(* Logix 5000 project; controller Google vendor 1 type 14 code 151 rev 31.11; software revision 31.00; part 4 of 5 *)
(* tags used below, declared in another part *)
   Infeed_Active : BOOL;
   L1_Clear_Out : BOOL;
   L1_Empty_Delay : TIMER;
   L1_Full_Delay : TIMER;
   L1_Zone1 : Zone_Data;
   L1_Zone1_2_ProdCode : DINT;
   L1_Zone1_2_ProdName : STRING;
   L1_Zone1_FWD : BOOL;
   L1_Zone1_PE : BOOL;
   L1_Zone1_ProdCode : DINT;
   L1_Zone1_ProdName : STRING;
   L1_Zone1_REV : BOOL;
   L1_Zone2 : Zone_Data;
   L1_Zone2_3_ProdCode : DINT;
   L1_Zone2_3_ProdName : STRING;
   L1_Zone2_FWD : BOOL;
   L1_Zone2_PE : BOOL;
   L1_Zone2_ProdCode : DINT;
   L1_Zone2_ProdName : STRING;
   L1_Zone2_REV : BOOL;
   L1_Zone3 : Zone_Data;
   L1_Zone3_4_ProdCode : DINT;
   L1_Zone3_4_ProdName : STRING;
   L1_Zone3_FWD : BOOL;
   L1_Zone3_PE : BOOL;
   L1_Zone3_ProdCode : DINT;
   L1_Zone3_ProdName : STRING;
   L1_Zone3_REV : BOOL;
   L1_Zone4 : End_Zone_Data;
   L1_Zone4_FWD : BOOL;
   L1_Zone4_PE : BOOL;
   L1_Zone4_ProdCode : DINT;
   L1_Zone4_ProdName : STRING;
   L1_Zone4_REV : BOOL;
   L1_Zone_Timeout : TIMER[8];
   L2_Empty_Delay : TIMER;
   L2_Full_Delay : TIMER;
   L2_Z1_Outfeed : BOOL;
   L2_Z2_Outfeed : BOOL;
   L2_Z3_Outfeed : BOOL;
   L2_Z4_Outfeed : BOOL;
   L2_Zone1 : Zone_Data;
   L2_Zone1_2_ProdCode : DINT;
   L2_Zone1_2_ProdName : STRING;
   L2_Zone1_FWD : BOOL;
   L2_Zone1_PE : BOOL;
   L2_Zone1_ProdCode : DINT;
   L2_Zone1_ProdName : STRING;
   L2_Zone1_REV : BOOL;
   L2_Zone2 : Zone_Data;
   L2_Zone2_3_ProdCode : DINT;
   L2_Zone2_3_ProdName : STRING;
   L2_Zone2_FWD : BOOL;
   L2_Zone2_PE : BOOL;
   L2_Zone2_ProdCode : DINT;
   L2_Zone2_ProdName : STRING;
   L2_Zone2_REV : BOOL;
   L2_Zone3 : Zone_Data;
   L2_Zone3_4_ProdCode : DINT;
   L2_Zone3_4_ProdName : STRING;
   L2_Zone3_FWD : BOOL;
   L2_Zone3_PE : BOOL;
   L2_Zone3_ProdCode : DINT;
   L2_Zone3_ProdName : STRING;
   L2_Zone3_REV : BOOL;
   L2_Zone4 : End_Zone_Data;
   L2_Zone4_FWD : BOOL;
   L2_Zone4_PE : BOOL;
   L2_Zone4_ProdCode : DINT;
   L2_Zone4_ProdName : STRING;
   L2_Zone4_REV : BOOL;
   L2_Zone_Timeout : TIMER[8];
   L3_Empty_Delay : TIMER;
   L3_Full_Delay : TIMER;
   L3_Z1_Outfeed : BOOL;
   L3_Z2_Outfeed : BOOL;
   L3_Z3_Outfeed : BOOL;
   L3_Z4_Outfeed : BOOL;
   L3_Zone1 : Zone_Data;
   L3_Zone1_2_ProdCode : DINT;
   L3_Zone1_2_ProdName : STRING;
   L3_Zone1_FWD : BOOL;
   L3_Zone1_PE : BOOL;
   L3_Zone1_ProdCode : DINT;
   L3_Zone1_ProdName : STRING;
   L3_Zone1_REV : BOOL;
   L3_Zone2 : Zone_Data;
   L3_Zone2_3_ProdCode : DINT;
   L3_Zone2_3_ProdName : STRING;
   L3_Zone2_FWD : BOOL;
   L3_Zone2_PE : BOOL;
   L3_Zone2_ProdCode : DINT;
   L3_Zone2_ProdName : STRING;
   L3_Zone2_REV : BOOL;
   L3_Zone3 : Zone_Data;
   L3_Zone3_4_ProdCode : DINT;
   L3_Zone3_4_ProdName : STRING;
   L3_Zone3_FWD : BOOL;
   L3_Zone3_PE : BOOL;
   L3_Zone3_ProdCode : DINT;
   L3_Zone3_ProdName : STRING;
   L3_Zone3_REV : BOOL;
   L3_Zone4 : End_Zone_Data;
   L3_Zone4_FWD : BOOL;
   L3_Zone4_PE : BOOL;
   L3_Zone4_ProdCode : DINT;
   L3_Zone4_ProdName : STRING;
   L3_Zone4_REV : BOOL;
   L3_Zone_Timeout : TIMER[8];
   L4_Empty_Delay : TIMER;
   L4_Full_Delay : TIMER;
   L4_Z1_Outfeed : BOOL;
   L4_Z2_Outfeed : BOOL;
   L4_Z3_Outfeed : BOOL;
   L4_Z4_Outfeed : BOOL;
   L4_Zone1 : Zone_Data;
   L4_Zone1_2_ProdCode : DINT;
   L4_Zone1_2_ProdName : STRING;
   L4_Zone1_FWD : BOOL;
   L4_Zone1_PE : BOOL;
   L4_Zone1_ProdCode : DINT;
   L4_Zone1_ProdName : STRING;
   L4_Zone1_REV : BOOL;
   L4_Zone2 : Zone_Data;
   L4_Zone2_3_ProdCode : DINT;
   L4_Zone2_3_ProdName : STRING;
   L4_Zone2_FWD : BOOL;
   L4_Zone2_PE : BOOL;
   L4_Zone2_ProdCode : DINT;
   L4_Zone2_ProdName : STRING;
   L4_Zone2_REV : BOOL;
   L4_Zone3 : Zone_Data;
   L4_Zone3_4_ProdCode : DINT;
   L4_Zone3_4_ProdName : STRING;
   L4_Zone3_FWD : BOOL;
   L4_Zone3_PE : BOOL;
   L4_Zone3_ProdCode : DINT;
   L4_Zone3_ProdName : STRING;
   L4_Zone3_REV : BOOL;
   L4_Zone4 : End_Zone_Data;
   L4_Zone4_FWD : BOOL;
   L4_Zone4_PE : BOOL;
   L4_Zone4_ProdCode : DINT;
   L4_Zone4_ProdName : STRING;
   L4_Zone4_REV : BOOL;
   L4_Zone_Timeout : TIMER[8];
   Level_1_Empty : BOOL;
   Level_1_Full : BOOL;
   Level_2_Empty : BOOL;
   Level_2_Full : BOOL;
   Level_3_Empty : BOOL;
   Level_3_Full : BOOL;
   Level_4_Empty : BOOL;
   Level_4_Full : BOOL;
   Lift_Current_Level : DINT;
   Lift_Required_Level : DINT;
   Lift_Zone : Lift_Zone_Data;
   LiftZone_FWD : BOOL;
   LiftZoneDownstream_ProdCode : DINT;
   LiftZoneDownstream_ProdName : STRING;
   Outfeed_Active : BOOL;
   Sort_Number : DINT;
(* MainProgram, continued *)

ROUTINE R09_L1_Conveyor   (* ladder *)
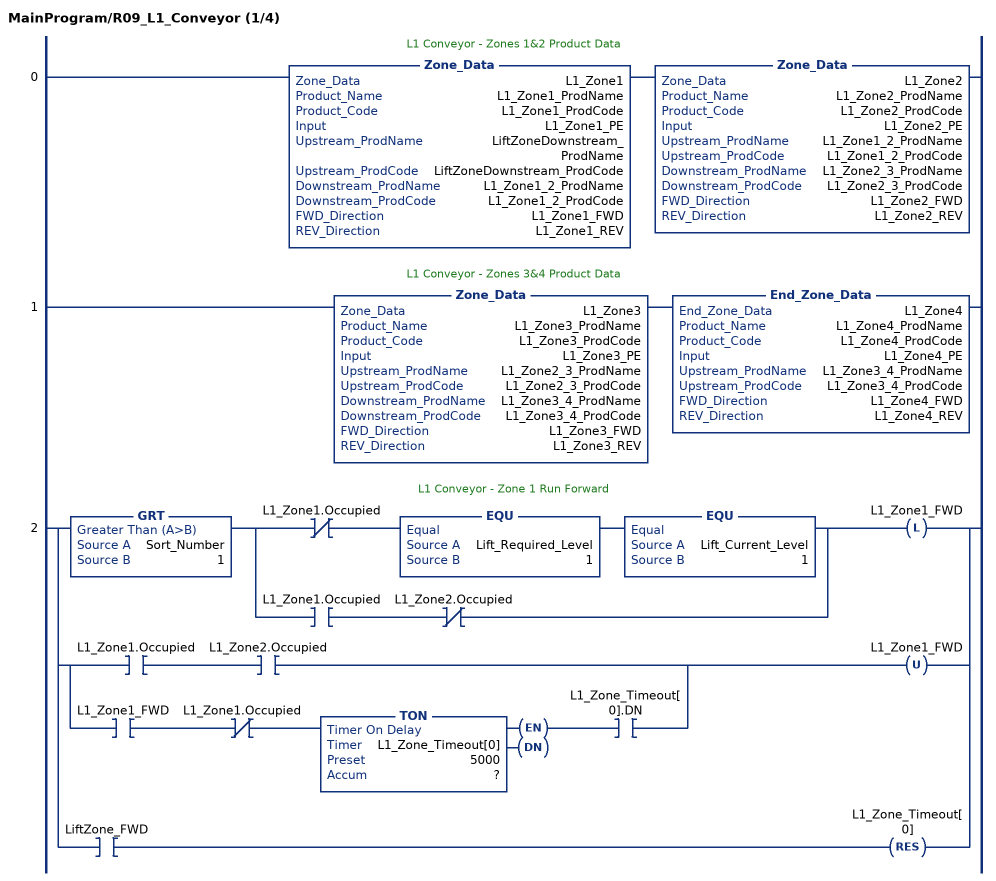
   // L1 Conveyor - Zones 1&2 Product Data
   0: Zone_Data(L1_Zone1,L1_Zone1_ProdName,L1_Zone1_ProdCode,L1_Zone1_PE,LiftZoneDownstream_ProdName,LiftZoneDownstream_ProdCode,L1_Zone1_2_ProdName,L1_Zone1_2_ProdCode,L1_Zone1_FWD,L1_Zone1_REV)Zone_Data(L1_Zone2,L1_Zone2_ProdName,L1_Zone2_ProdCode,L1_Zone2_PE,L1_Zone1_2_ProdName,L1_Zone1_2_ProdCode,L1_Zone2_3_ProdName,L1_Zone2_3_ProdCode,L1_Zone2_FWD,L1_Zone2_REV);
   // L1 Conveyor - Zones 3&4 Product Data
   1: Zone_Data(L1_Zone3,L1_Zone3_ProdName,L1_Zone3_ProdCode,L1_Zone3_PE,L1_Zone2_3_ProdName,L1_Zone2_3_ProdCode,L1_Zone3_4_ProdName,L1_Zone3_4_ProdCode,L1_Zone3_FWD,L1_Zone3_REV)End_Zone_Data(L1_Zone4,L1_Zone4_ProdName,L1_Zone4_ProdCode,L1_Zone4_PE,L1_Zone3_4_ProdName,L1_Zone3_4_ProdCode,L1_Zone4_FWD,L1_Zone4_REV);
   // L1 Conveyor - Zone 1 Run Forward
   2: [GRT(Sort_Number,1) [XIO(L1_Zone1.Occupied) EQU(Lift_Required_Level,1) EQU(Lift_Current_Level,1) ,XIC(L1_Zone1.Occupied) XIO(L1_Zone2.Occupied) ] OTL(L1_Zone1_FWD) ,[XIC(L1_Zone1.Occupied) XIC(L1_Zone2.Occupied) ,XIC(L1_Zone1_FWD) XIO(L1_Zone1.Occupied) TON(L1_Zone_Timeout[0],?,?) XIC(L1_Zone_Timeout[0].DN) ] OTU(L1_Zone1_FWD) ,XIC(LiftZone_FWD) RES(L1_Zone_Timeout[0]) ];
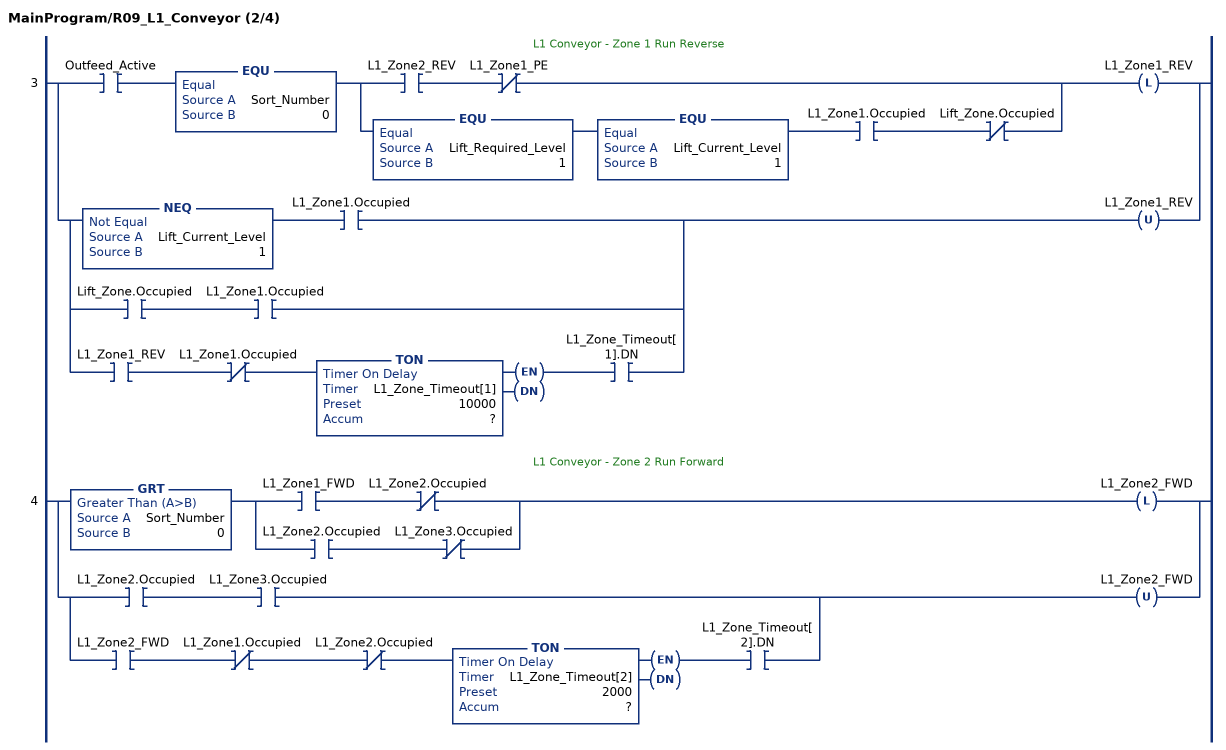
   // L1 Conveyor - Zone 1 Run Reverse
   3: [XIC(Outfeed_Active) EQU(Sort_Number,0) [XIC(L1_Zone2_REV) XIO(L1_Zone1_PE) ,EQU(Lift_Required_Level,1) EQU(Lift_Current_Level,1) XIC(L1_Zone1.Occupied) XIO(Lift_Zone.Occupied) ] OTL(L1_Zone1_REV) ,[NEQ(Lift_Current_Level,1) XIC(L1_Zone1.Occupied) ,XIC(Lift_Zone.Occupied) XIC(L1_Zone1.Occupied) ,XIC(L1_Zone1_REV) XIO(L1_Zone1.Occupied) TON(L1_Zone_Timeout[1],?,?) XIC(L1_Zone_Timeout[1].DN) ] OTU(L1_Zone1_REV) ];
   // L1 Conveyor - Zone 2 Run Forward
   4: [GRT(Sort_Number,0) [XIC(L1_Zone1_FWD) XIO(L1_Zone2.Occupied) ,XIC(L1_Zone2.Occupied) XIO(L1_Zone3.Occupied) ] OTL(L1_Zone2_FWD) ,[XIC(L1_Zone2.Occupied) XIC(L1_Zone3.Occupied) ,XIC(L1_Zone2_FWD) XIO(L1_Zone1.Occupied) XIO(L1_Zone2.Occupied) TON(L1_Zone_Timeout[2],?,?) XIC(L1_Zone_Timeout[2].DN) ] OTU(L1_Zone2_FWD) ];
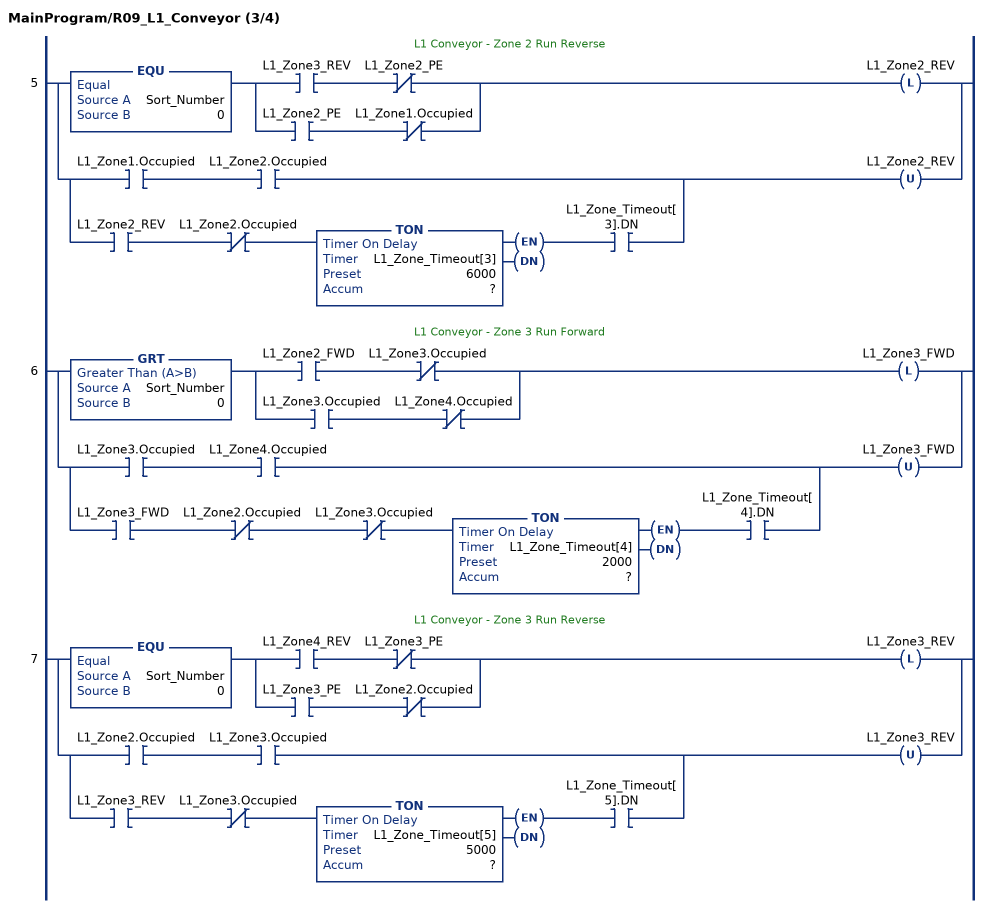
   // L1 Conveyor - Zone 2 Run Reverse
   5: [EQU(Sort_Number,0) [XIC(L1_Zone3_REV) XIO(L1_Zone2_PE) ,XIC(L1_Zone2_PE) XIO(L1_Zone1.Occupied) ] OTL(L1_Zone2_REV) ,[XIC(L1_Zone1.Occupied) XIC(L1_Zone2.Occupied) ,XIC(L1_Zone2_REV) XIO(L1_Zone2.Occupied) TON(L1_Zone_Timeout[3],?,?) XIC(L1_Zone_Timeout[3].DN) ] OTU(L1_Zone2_REV) ];
   // L1 Conveyor - Zone 3 Run Forward
   6: [GRT(Sort_Number,0) [XIC(L1_Zone2_FWD) XIO(L1_Zone3.Occupied) ,XIC(L1_Zone3.Occupied) XIO(L1_Zone4.Occupied) ] OTL(L1_Zone3_FWD) ,[XIC(L1_Zone3.Occupied) XIC(L1_Zone4.Occupied) ,XIC(L1_Zone3_FWD) XIO(L1_Zone2.Occupied) XIO(L1_Zone3.Occupied) TON(L1_Zone_Timeout[4],?,?) XIC(L1_Zone_Timeout[4].DN) ] OTU(L1_Zone3_FWD) ];
   // L1 Conveyor - Zone 3 Run Reverse
   7: [EQU(Sort_Number,0) [XIC(L1_Zone4_REV) XIO(L1_Zone3_PE) ,XIC(L1_Zone3_PE) XIO(L1_Zone2.Occupied) ] OTL(L1_Zone3_REV) ,[XIC(L1_Zone2.Occupied) XIC(L1_Zone3.Occupied) ,XIC(L1_Zone3_REV) XIO(L1_Zone3.Occupied) TON(L1_Zone_Timeout[5],?,?) XIC(L1_Zone_Timeout[5].DN) ] OTU(L1_Zone3_REV) ];
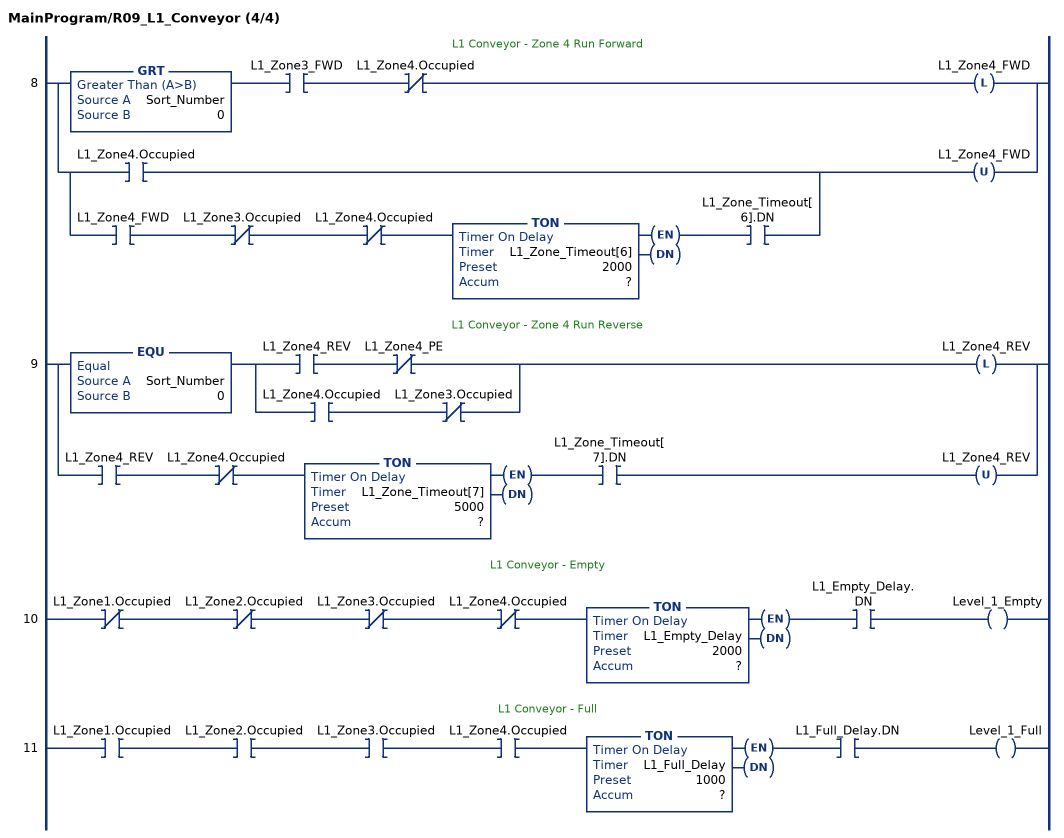
   // L1 Conveyor - Zone 4 Run Forward
   8: [GRT(Sort_Number,0) XIC(L1_Zone3_FWD) XIO(L1_Zone4.Occupied) OTL(L1_Zone4_FWD) ,[XIC(L1_Zone4.Occupied) ,XIC(L1_Zone4_FWD) XIO(L1_Zone3.Occupied) XIO(L1_Zone4.Occupied) TON(L1_Zone_Timeout[6],?,?) XIC(L1_Zone_Timeout[6].DN) ] OTU(L1_Zone4_FWD) ];
   // L1 Conveyor - Zone 4 Run Reverse
   9: [EQU(Sort_Number,0) [XIC(L1_Zone4_REV) XIO(L1_Zone4_PE) ,XIC(L1_Zone4.Occupied) XIO(L1_Zone3.Occupied) ] OTL(L1_Zone4_REV) ,XIC(L1_Zone4_REV) XIO(L1_Zone4.Occupied) TON(L1_Zone_Timeout[7],?,?) XIC(L1_Zone_Timeout[7].DN) OTU(L1_Zone4_REV) ];
   // L1 Conveyor - Empty
   10: XIO(L1_Zone1.Occupied)XIO(L1_Zone2.Occupied)XIO(L1_Zone3.Occupied)XIO(L1_Zone4.Occupied)TON(L1_Empty_Delay,?,?)XIC(L1_Empty_Delay.DN)OTE(Level_1_Empty);
   // L1 Conveyor - Full
   11: XIC(L1_Zone1.Occupied)XIC(L1_Zone2.Occupied)XIC(L1_Zone3.Occupied)XIC(L1_Zone4.Occupied)TON(L1_Full_Delay,?,?)XIC(L1_Full_Delay.DN)OTE(Level_1_Full);
END_ROUTINE

ROUTINE R10_L2_Conveyor   (* ladder *)
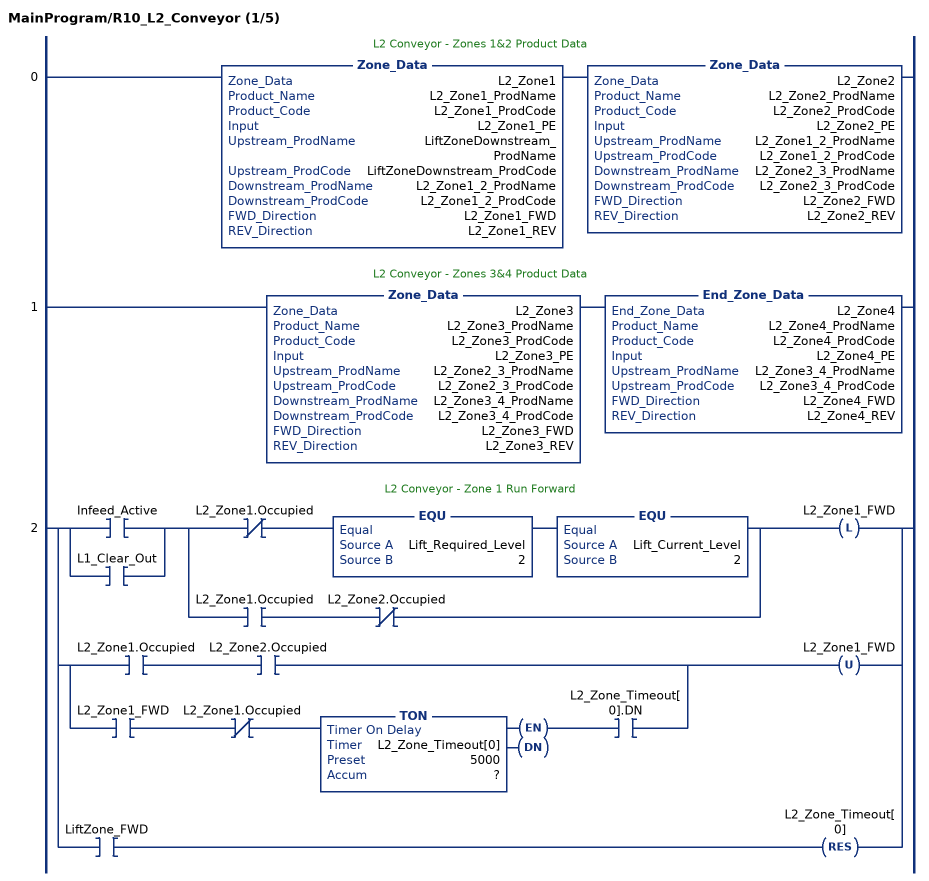
   // L2 Conveyor - Zones 1&2 Product Data
   0: Zone_Data(L2_Zone1,L2_Zone1_ProdName,L2_Zone1_ProdCode,L2_Zone1_PE,LiftZoneDownstream_ProdName,LiftZoneDownstream_ProdCode,L2_Zone1_2_ProdName,L2_Zone1_2_ProdCode,L2_Zone1_FWD,L2_Zone1_REV)Zone_Data(L2_Zone2,L2_Zone2_ProdName,L2_Zone2_ProdCode,L2_Zone2_PE,L2_Zone1_2_ProdName,L2_Zone1_2_ProdCode,L2_Zone2_3_ProdName,L2_Zone2_3_ProdCode,L2_Zone2_FWD,L2_Zone2_REV);
   // L2 Conveyor - Zones 3&4 Product Data
   1: Zone_Data(L2_Zone3,L2_Zone3_ProdName,L2_Zone3_ProdCode,L2_Zone3_PE,L2_Zone2_3_ProdName,L2_Zone2_3_ProdCode,L2_Zone3_4_ProdName,L2_Zone3_4_ProdCode,L2_Zone3_FWD,L2_Zone3_REV)End_Zone_Data(L2_Zone4,L2_Zone4_ProdName,L2_Zone4_ProdCode,L2_Zone4_PE,L2_Zone3_4_ProdName,L2_Zone3_4_ProdCode,L2_Zone4_FWD,L2_Zone4_REV);
   // L2 Conveyor - Zone 1 Run Forward
   2: [[XIC(Infeed_Active) ,XIC(L1_Clear_Out) ] [XIO(L2_Zone1.Occupied) EQU(Lift_Required_Level,2) EQU(Lift_Current_Level,2) ,XIC(L2_Zone1.Occupied) XIO(L2_Zone2.Occupied) ] OTL(L2_Zone1_FWD) ,[XIC(L2_Zone1.Occupied) XIC(L2_Zone2.Occupied) ,XIC(L2_Zone1_FWD) XIO(L2_Zone1.Occupied) TON(L2_Zone_Timeout[0],?,?) XIC(L2_Zone_Timeout[0].DN) ] OTU(L2_Zone1_FWD) ,XIC(LiftZone_FWD) RES(L2_Zone_Timeout[0]) ];
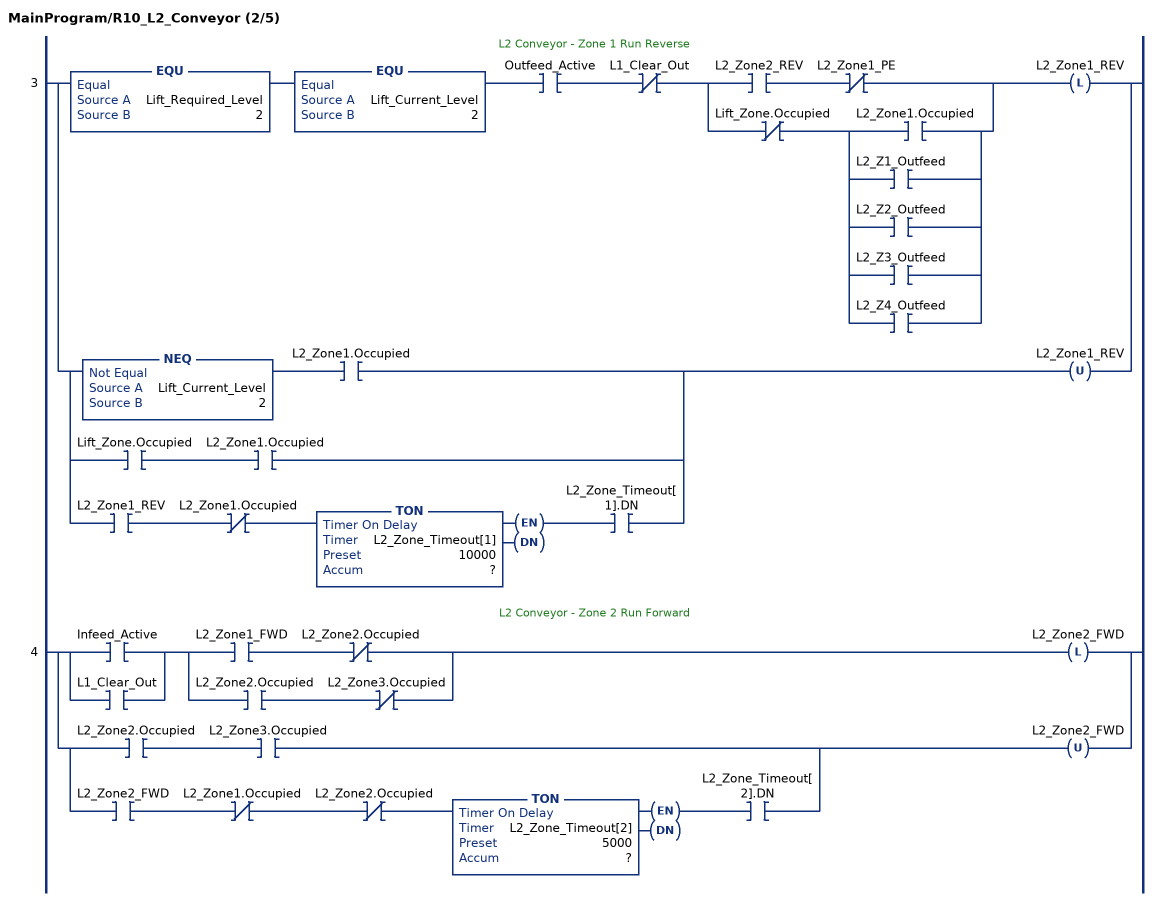
   // L2 Conveyor - Zone 1 Run Reverse
   3: [EQU(Lift_Required_Level,2) EQU(Lift_Current_Level,2) XIC(Outfeed_Active) XIO(L1_Clear_Out) [XIC(L2_Zone2_REV) XIO(L2_Zone1_PE) ,XIO(Lift_Zone.Occupied) [XIC(L2_Zone1.Occupied) ,XIC(L2_Z1_Outfeed) ,XIC(L2_Z2_Outfeed) ,XIC(L2_Z3_Outfeed) ,XIC(L2_Z4_Outfeed) ] ] OTL(L2_Zone1_REV) ,[NEQ(Lift_Current_Level,2) XIC(L2_Zone1.Occupied) ,XIC(Lift_Zone.Occupied) XIC(L2_Zone1.Occupied) ,XIC(L2_Zone1_REV) XIO(L2_Zone1.Occupied) TON(L2_Zone_Timeout[1],?,?) XIC(L2_Zone_Timeout[1].DN) ] OTU(L2_Zone1_REV) ];
   // L2 Conveyor - Zone 2 Run Forward
   4: [[XIC(Infeed_Active) ,XIC(L1_Clear_Out) ] [XIC(L2_Zone1_FWD) XIO(L2_Zone2.Occupied) ,XIC(L2_Zone2.Occupied) XIO(L2_Zone3.Occupied) ] OTL(L2_Zone2_FWD) ,[XIC(L2_Zone2.Occupied) XIC(L2_Zone3.Occupied) ,XIC(L2_Zone2_FWD) XIO(L2_Zone1.Occupied) XIO(L2_Zone2.Occupied) TON(L2_Zone_Timeout[2],?,?) XIC(L2_Zone_Timeout[2].DN) ] OTU(L2_Zone2_FWD) ];
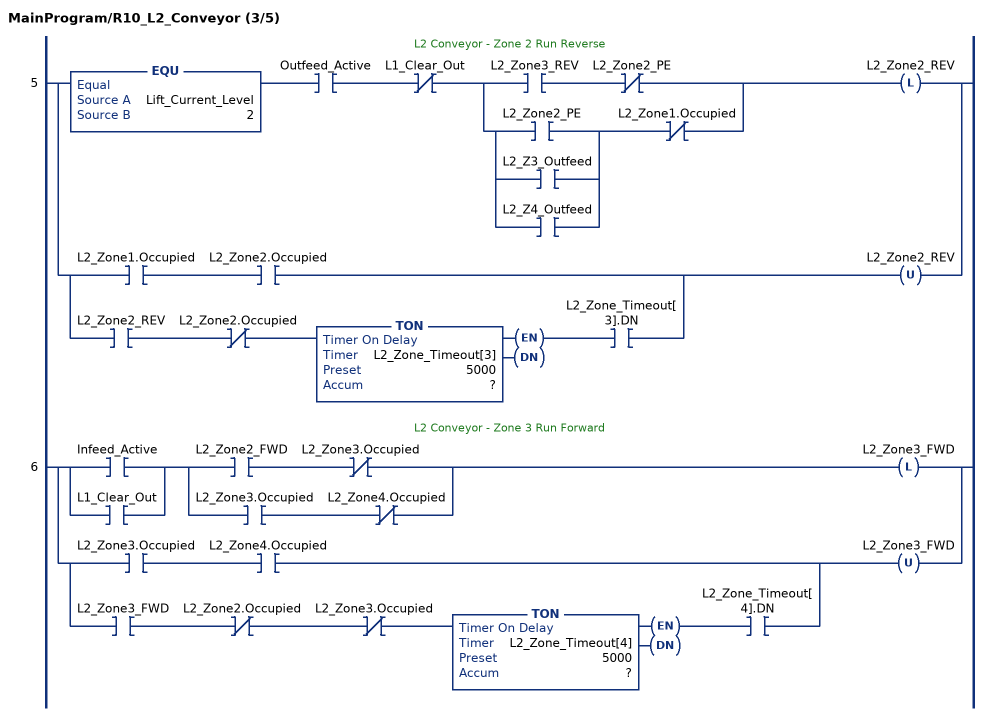
   // L2 Conveyor - Zone 2 Run Reverse
   5: [EQU(Lift_Current_Level,2) XIC(Outfeed_Active) XIO(L1_Clear_Out) [XIC(L2_Zone3_REV) XIO(L2_Zone2_PE) ,[XIC(L2_Zone2_PE) ,XIC(L2_Z3_Outfeed) ,XIC(L2_Z4_Outfeed) ] XIO(L2_Zone1.Occupied) ] OTL(L2_Zone2_REV) ,[XIC(L2_Zone1.Occupied) XIC(L2_Zone2.Occupied) ,XIC(L2_Zone2_REV) XIO(L2_Zone2.Occupied) TON(L2_Zone_Timeout[3],?,?) XIC(L2_Zone_Timeout[3].DN) ] OTU(L2_Zone2_REV) ];
   // L2 Conveyor - Zone 3 Run Forward
   6: [[XIC(Infeed_Active) ,XIC(L1_Clear_Out) ] [XIC(L2_Zone2_FWD) XIO(L2_Zone3.Occupied) ,XIC(L2_Zone3.Occupied) XIO(L2_Zone4.Occupied) ] OTL(L2_Zone3_FWD) ,[XIC(L2_Zone3.Occupied) XIC(L2_Zone4.Occupied) ,XIC(L2_Zone3_FWD) XIO(L2_Zone2.Occupied) XIO(L2_Zone3.Occupied) TON(L2_Zone_Timeout[4],?,?) XIC(L2_Zone_Timeout[4].DN) ] OTU(L2_Zone3_FWD) ];
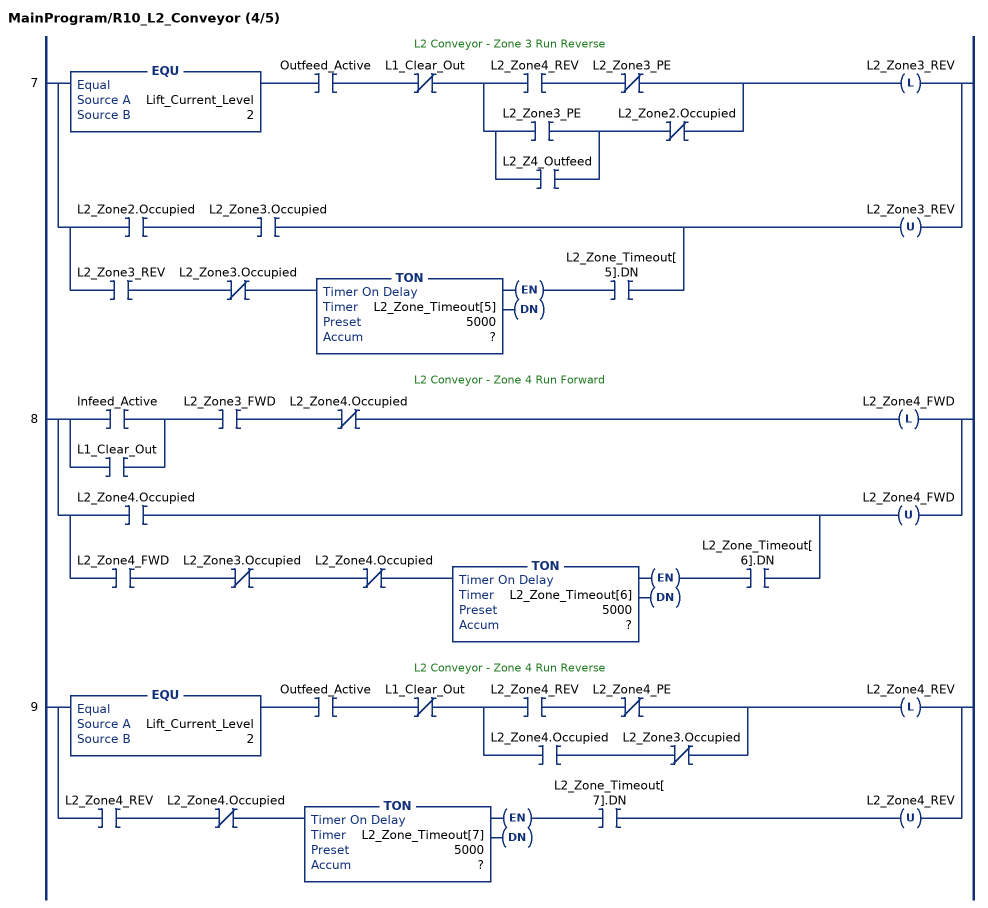
   // L2 Conveyor - Zone 3 Run Reverse
   7: [EQU(Lift_Current_Level,2) XIC(Outfeed_Active) XIO(L1_Clear_Out) [XIC(L2_Zone4_REV) XIO(L2_Zone3_PE) ,[XIC(L2_Zone3_PE) ,XIC(L2_Z4_Outfeed) ] XIO(L2_Zone2.Occupied) ] OTL(L2_Zone3_REV) ,[XIC(L2_Zone2.Occupied) XIC(L2_Zone3.Occupied) ,XIC(L2_Zone3_REV) XIO(L2_Zone3.Occupied) TON(L2_Zone_Timeout[5],?,?) XIC(L2_Zone_Timeout[5].DN) ] OTU(L2_Zone3_REV) ];
   // L2 Conveyor - Zone 4 Run Forward
   8: [[XIC(Infeed_Active) ,XIC(L1_Clear_Out) ] XIC(L2_Zone3_FWD) XIO(L2_Zone4.Occupied) OTL(L2_Zone4_FWD) ,[XIC(L2_Zone4.Occupied) ,XIC(L2_Zone4_FWD) XIO(L2_Zone3.Occupied) XIO(L2_Zone4.Occupied) TON(L2_Zone_Timeout[6],?,?) XIC(L2_Zone_Timeout[6].DN) ] OTU(L2_Zone4_FWD) ];
   // L2 Conveyor - Zone 4 Run Reverse
   9: [EQU(Lift_Current_Level,2) XIC(Outfeed_Active) XIO(L1_Clear_Out) [XIC(L2_Zone4_REV) XIO(L2_Zone4_PE) ,XIC(L2_Zone4.Occupied) XIO(L2_Zone3.Occupied) ] OTL(L2_Zone4_REV) ,XIC(L2_Zone4_REV) XIO(L2_Zone4.Occupied) TON(L2_Zone_Timeout[7],?,?) XIC(L2_Zone_Timeout[7].DN) OTU(L2_Zone4_REV) ];
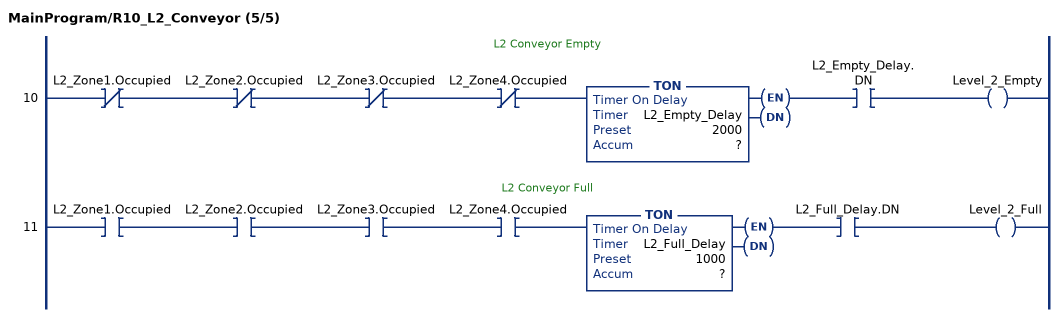
   // L2 Conveyor Empty
   10: XIO(L2_Zone1.Occupied)XIO(L2_Zone2.Occupied)XIO(L2_Zone3.Occupied)XIO(L2_Zone4.Occupied)TON(L2_Empty_Delay,?,?)XIC(L2_Empty_Delay.DN)OTE(Level_2_Empty);
   // L2 Conveyor Full
   11: XIC(L2_Zone1.Occupied)XIC(L2_Zone2.Occupied)XIC(L2_Zone3.Occupied)XIC(L2_Zone4.Occupied)TON(L2_Full_Delay,?,?)XIC(L2_Full_Delay.DN)OTE(Level_2_Full);
END_ROUTINE

ROUTINE R11_L3_Conveyor   (* ladder *)
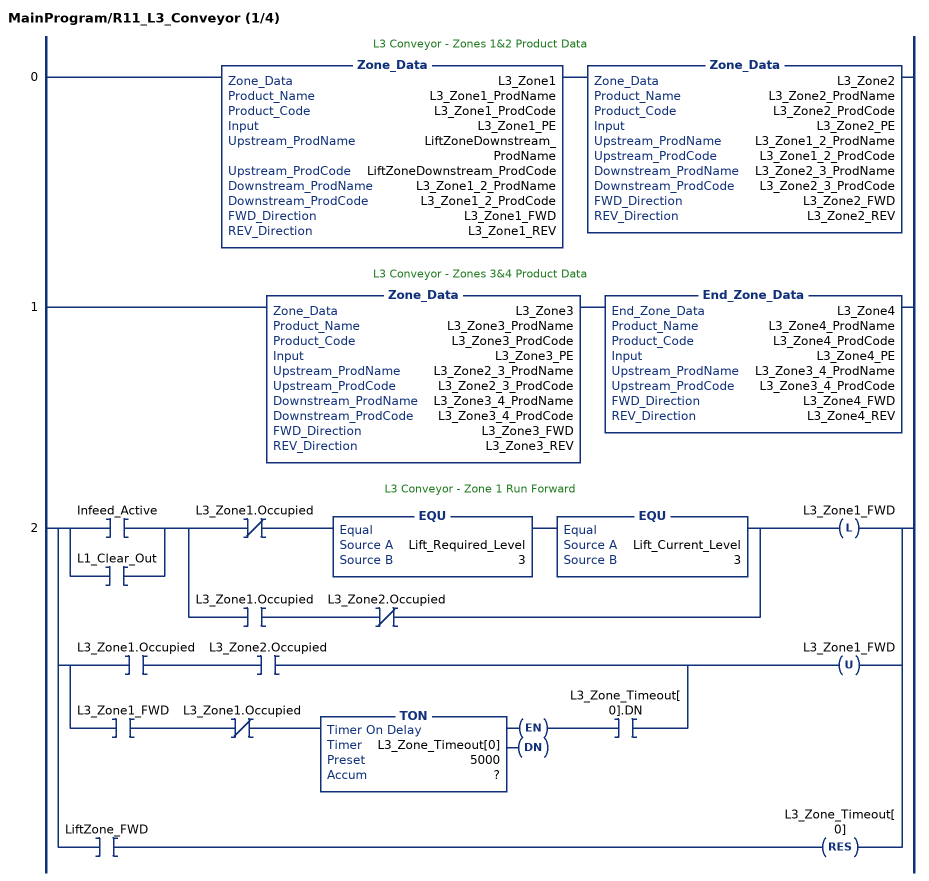
   // L3 Conveyor - Zones 1&2 Product Data
   0: Zone_Data(L3_Zone1,L3_Zone1_ProdName,L3_Zone1_ProdCode,L3_Zone1_PE,LiftZoneDownstream_ProdName,LiftZoneDownstream_ProdCode,L3_Zone1_2_ProdName,L3_Zone1_2_ProdCode,L3_Zone1_FWD,L3_Zone1_REV)Zone_Data(L3_Zone2,L3_Zone2_ProdName,L3_Zone2_ProdCode,L3_Zone2_PE,L3_Zone1_2_ProdName,L3_Zone1_2_ProdCode,L3_Zone2_3_ProdName,L3_Zone2_3_ProdCode,L3_Zone2_FWD,L3_Zone2_REV);
   // L3 Conveyor - Zones 3&4 Product Data
   1: Zone_Data(L3_Zone3,L3_Zone3_ProdName,L3_Zone3_ProdCode,L3_Zone3_PE,L3_Zone2_3_ProdName,L3_Zone2_3_ProdCode,L3_Zone3_4_ProdName,L3_Zone3_4_ProdCode,L3_Zone3_FWD,L3_Zone3_REV)End_Zone_Data(L3_Zone4,L3_Zone4_ProdName,L3_Zone4_ProdCode,L3_Zone4_PE,L3_Zone3_4_ProdName,L3_Zone3_4_ProdCode,L3_Zone4_FWD,L3_Zone4_REV);
   // L3 Conveyor - Zone 1 Run Forward
   2: [[XIC(Infeed_Active) ,XIC(L1_Clear_Out) ] [XIO(L3_Zone1.Occupied) EQU(Lift_Required_Level,3) EQU(Lift_Current_Level,3) ,XIC(L3_Zone1.Occupied) XIO(L3_Zone2.Occupied) ] OTL(L3_Zone1_FWD) ,[XIC(L3_Zone1.Occupied) XIC(L3_Zone2.Occupied) ,XIC(L3_Zone1_FWD) XIO(L3_Zone1.Occupied) TON(L3_Zone_Timeout[0],?,?) XIC(L3_Zone_Timeout[0].DN) ] OTU(L3_Zone1_FWD) ,XIC(LiftZone_FWD) RES(L3_Zone_Timeout[0]) ];
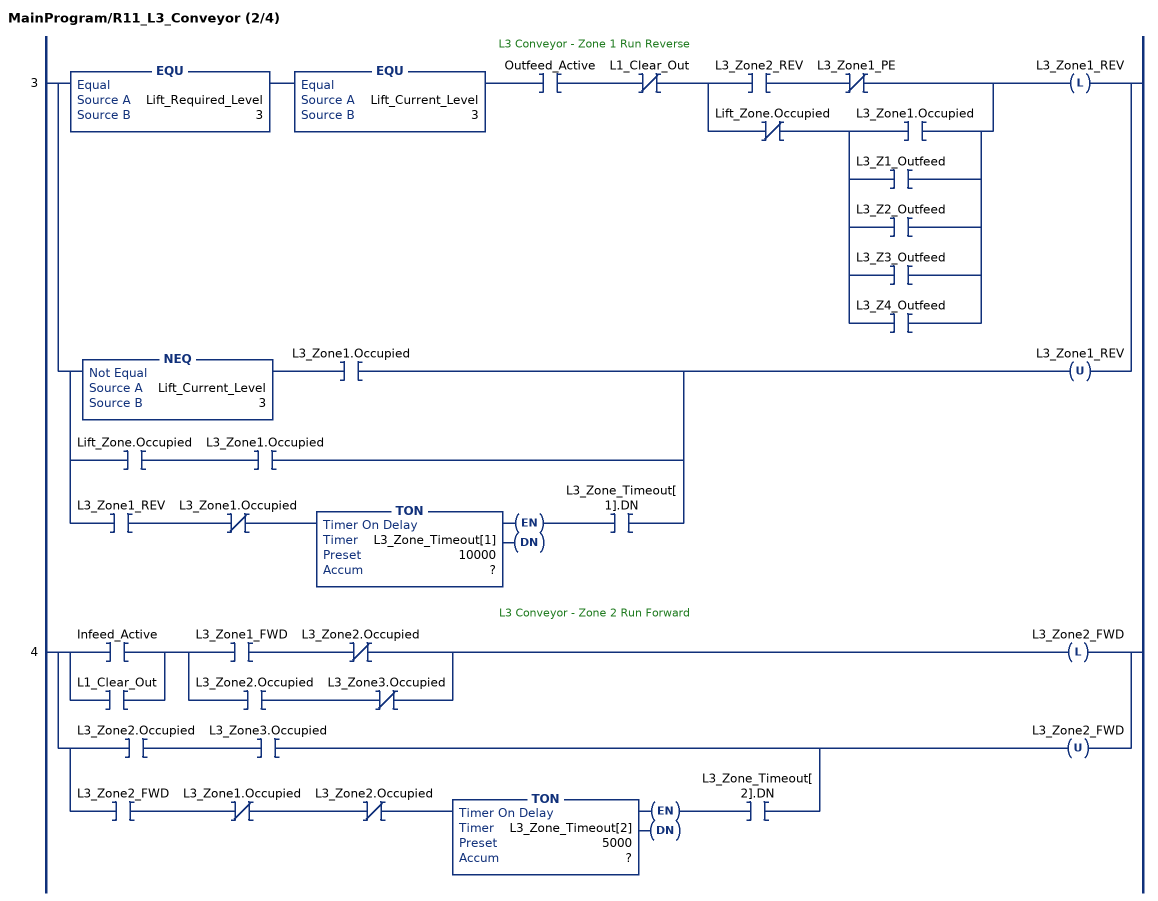
   // L3 Conveyor - Zone 1 Run Reverse
   3: [EQU(Lift_Required_Level,3) EQU(Lift_Current_Level,3) XIC(Outfeed_Active) XIO(L1_Clear_Out) [XIC(L3_Zone2_REV) XIO(L3_Zone1_PE) ,XIO(Lift_Zone.Occupied) [XIC(L3_Zone1.Occupied) ,XIC(L3_Z1_Outfeed) ,XIC(L3_Z2_Outfeed) ,XIC(L3_Z3_Outfeed) ,XIC(L3_Z4_Outfeed) ] ] OTL(L3_Zone1_REV) ,[NEQ(Lift_Current_Level,3) XIC(L3_Zone1.Occupied) ,XIC(Lift_Zone.Occupied) XIC(L3_Zone1.Occupied) ,XIC(L3_Zone1_REV) XIO(L3_Zone1.Occupied) TON(L3_Zone_Timeout[1],?,?) XIC(L3_Zone_Timeout[1].DN) ] OTU(L3_Zone1_REV) ];
   // L3 Conveyor - Zone 2 Run Forward
   4: [[XIC(Infeed_Active) ,XIC(L1_Clear_Out) ] [XIC(L3_Zone1_FWD) XIO(L3_Zone2.Occupied) ,XIC(L3_Zone2.Occupied) XIO(L3_Zone3.Occupied) ] OTL(L3_Zone2_FWD) ,[XIC(L3_Zone2.Occupied) XIC(L3_Zone3.Occupied) ,XIC(L3_Zone2_FWD) XIO(L3_Zone1.Occupied) XIO(L3_Zone2.Occupied) TON(L3_Zone_Timeout[2],?,?) XIC(L3_Zone_Timeout[2].DN) ] OTU(L3_Zone2_FWD) ];
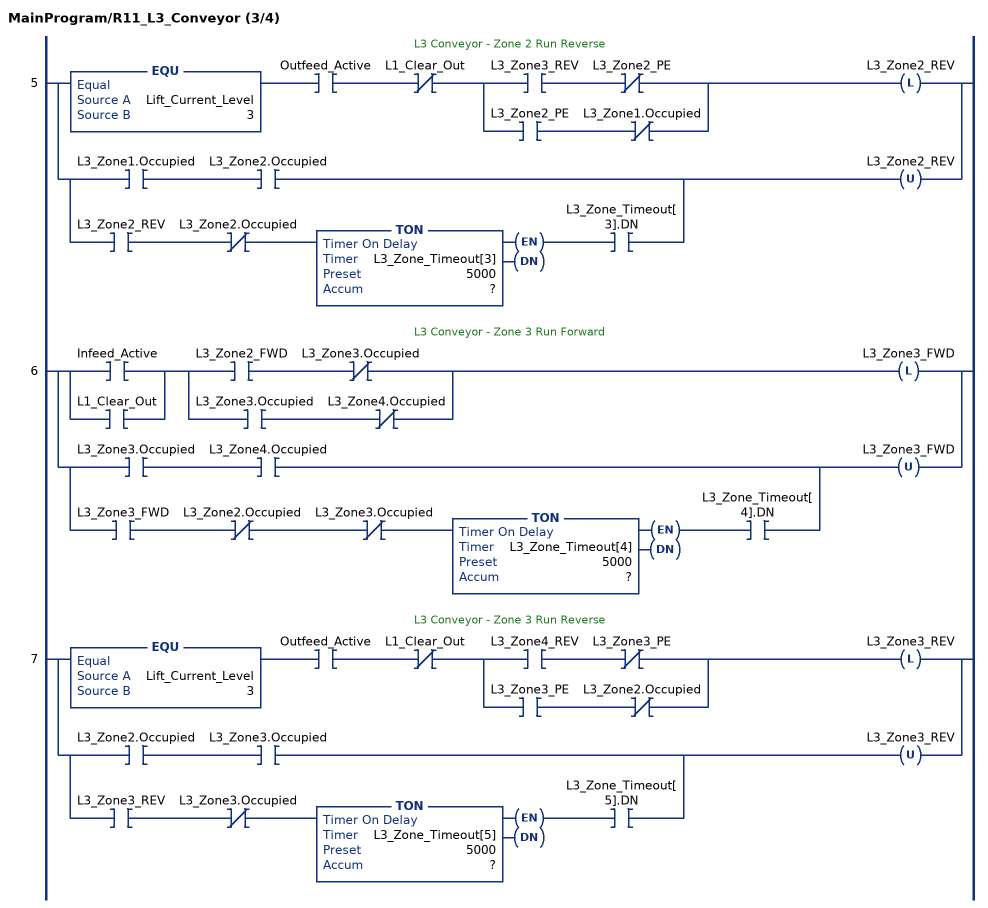
   // L3 Conveyor - Zone 2 Run Reverse
   5: [EQU(Lift_Current_Level,3) XIC(Outfeed_Active) XIO(L1_Clear_Out) [XIC(L3_Zone3_REV) XIO(L3_Zone2_PE) ,XIC(L3_Zone2_PE) XIO(L3_Zone1.Occupied) ] OTL(L3_Zone2_REV) ,[XIC(L3_Zone1.Occupied) XIC(L3_Zone2.Occupied) ,XIC(L3_Zone2_REV) XIO(L3_Zone2.Occupied) TON(L3_Zone_Timeout[3],?,?) XIC(L3_Zone_Timeout[3].DN) ] OTU(L3_Zone2_REV) ];
   // L3 Conveyor - Zone 3 Run Forward
   6: [[XIC(Infeed_Active) ,XIC(L1_Clear_Out) ] [XIC(L3_Zone2_FWD) XIO(L3_Zone3.Occupied) ,XIC(L3_Zone3.Occupied) XIO(L3_Zone4.Occupied) ] OTL(L3_Zone3_FWD) ,[XIC(L3_Zone3.Occupied) XIC(L3_Zone4.Occupied) ,XIC(L3_Zone3_FWD) XIO(L3_Zone2.Occupied) XIO(L3_Zone3.Occupied) TON(L3_Zone_Timeout[4],?,?) XIC(L3_Zone_Timeout[4].DN) ] OTU(L3_Zone3_FWD) ];
   // L3 Conveyor - Zone 3 Run Reverse
   7: [EQU(Lift_Current_Level,3) XIC(Outfeed_Active) XIO(L1_Clear_Out) [XIC(L3_Zone4_REV) XIO(L3_Zone3_PE) ,XIC(L3_Zone3_PE) XIO(L3_Zone2.Occupied) ] OTL(L3_Zone3_REV) ,[XIC(L3_Zone2.Occupied) XIC(L3_Zone3.Occupied) ,XIC(L3_Zone3_REV) XIO(L3_Zone3.Occupied) TON(L3_Zone_Timeout[5],?,?) XIC(L3_Zone_Timeout[5].DN) ] OTU(L3_Zone3_REV) ];
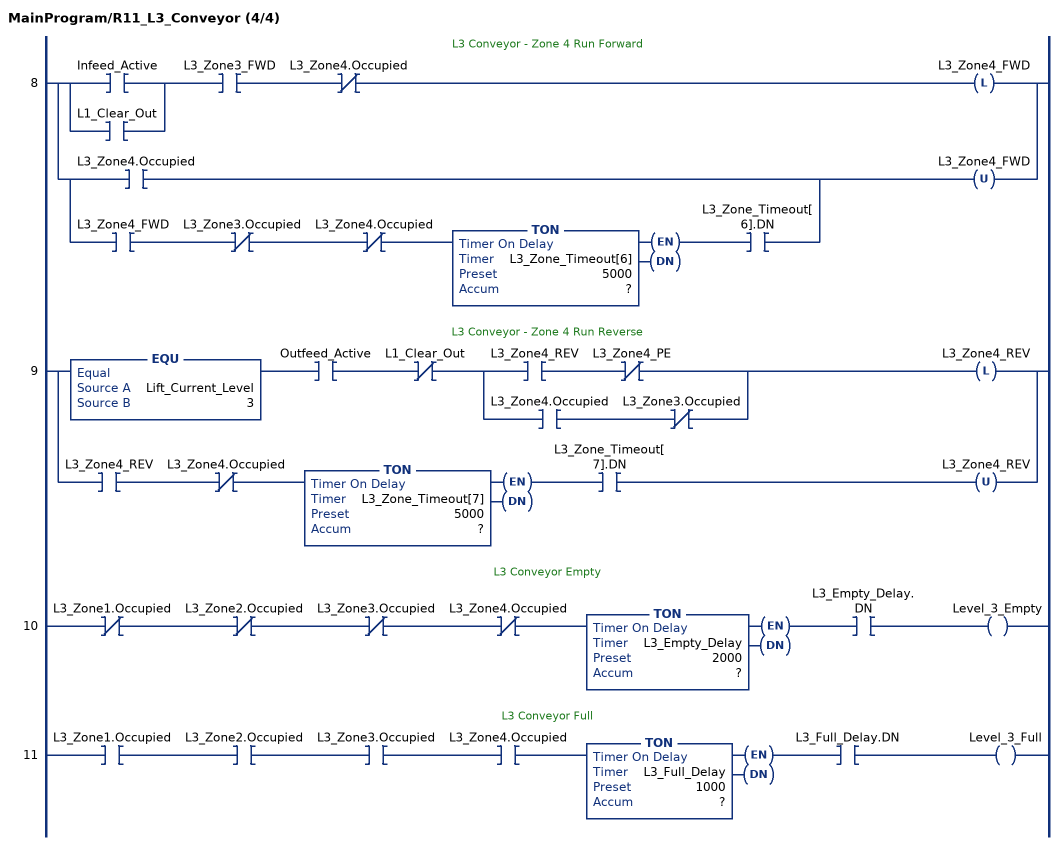
   // L3 Conveyor - Zone 4 Run Forward
   8: [[XIC(Infeed_Active) ,XIC(L1_Clear_Out) ] XIC(L3_Zone3_FWD) XIO(L3_Zone4.Occupied) OTL(L3_Zone4_FWD) ,[XIC(L3_Zone4.Occupied) ,XIC(L3_Zone4_FWD) XIO(L3_Zone3.Occupied) XIO(L3_Zone4.Occupied) TON(L3_Zone_Timeout[6],?,?) XIC(L3_Zone_Timeout[6].DN) ] OTU(L3_Zone4_FWD) ];
   // L3 Conveyor - Zone 4 Run Reverse
   9: [EQU(Lift_Current_Level,3) XIC(Outfeed_Active) XIO(L1_Clear_Out) [XIC(L3_Zone4_REV) XIO(L3_Zone4_PE) ,XIC(L3_Zone4.Occupied) XIO(L3_Zone3.Occupied) ] OTL(L3_Zone4_REV) ,XIC(L3_Zone4_REV) XIO(L3_Zone4.Occupied) TON(L3_Zone_Timeout[7],?,?) XIC(L3_Zone_Timeout[7].DN) OTU(L3_Zone4_REV) ];
   // L3 Conveyor Empty
   10: XIO(L3_Zone1.Occupied)XIO(L3_Zone2.Occupied)XIO(L3_Zone3.Occupied)XIO(L3_Zone4.Occupied)TON(L3_Empty_Delay,?,?)XIC(L3_Empty_Delay.DN)OTE(Level_3_Empty);
   // L3 Conveyor Full
   11: XIC(L3_Zone1.Occupied)XIC(L3_Zone2.Occupied)XIC(L3_Zone3.Occupied)XIC(L3_Zone4.Occupied)TON(L3_Full_Delay,?,?)XIC(L3_Full_Delay.DN)OTE(Level_3_Full);
END_ROUTINE

ROUTINE R12_L4_Conveyor   (* ladder *)
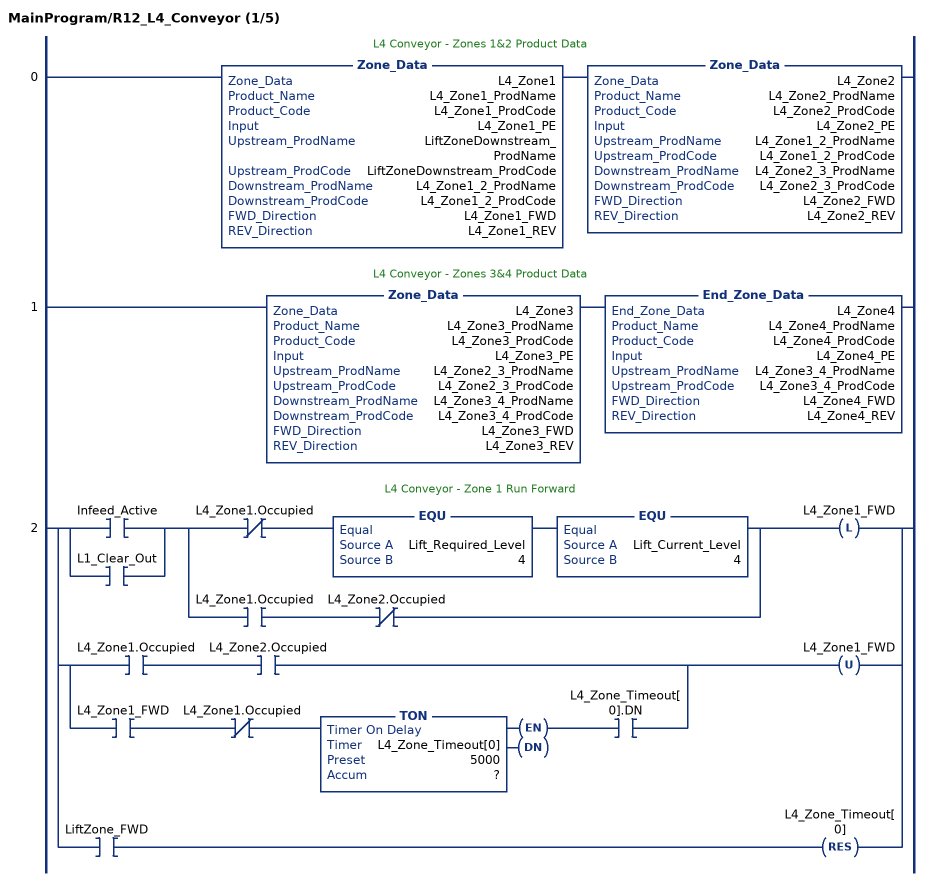
   // L4 Conveyor - Zones 1&2 Product Data
   0: Zone_Data(L4_Zone1,L4_Zone1_ProdName,L4_Zone1_ProdCode,L4_Zone1_PE,LiftZoneDownstream_ProdName,LiftZoneDownstream_ProdCode,L4_Zone1_2_ProdName,L4_Zone1_2_ProdCode,L4_Zone1_FWD,L4_Zone1_REV)Zone_Data(L4_Zone2,L4_Zone2_ProdName,L4_Zone2_ProdCode,L4_Zone2_PE,L4_Zone1_2_ProdName,L4_Zone1_2_ProdCode,L4_Zone2_3_ProdName,L4_Zone2_3_ProdCode,L4_Zone2_FWD,L4_Zone2_REV);
   // L4 Conveyor - Zones 3&4 Product Data
   1: Zone_Data(L4_Zone3,L4_Zone3_ProdName,L4_Zone3_ProdCode,L4_Zone3_PE,L4_Zone2_3_ProdName,L4_Zone2_3_ProdCode,L4_Zone3_4_ProdName,L4_Zone3_4_ProdCode,L4_Zone3_FWD,L4_Zone3_REV)End_Zone_Data(L4_Zone4,L4_Zone4_ProdName,L4_Zone4_ProdCode,L4_Zone4_PE,L4_Zone3_4_ProdName,L4_Zone3_4_ProdCode,L4_Zone4_FWD,L4_Zone4_REV);
   // L4 Conveyor - Zone 1 Run Forward
   2: [[XIC(Infeed_Active) ,XIC(L1_Clear_Out) ] [XIO(L4_Zone1.Occupied) EQU(Lift_Required_Level,4) EQU(Lift_Current_Level,4) ,XIC(L4_Zone1.Occupied) XIO(L4_Zone2.Occupied) ] OTL(L4_Zone1_FWD) ,[XIC(L4_Zone1.Occupied) XIC(L4_Zone2.Occupied) ,XIC(L4_Zone1_FWD) XIO(L4_Zone1.Occupied) TON(L4_Zone_Timeout[0],?,?) XIC(L4_Zone_Timeout[0].DN) ] OTU(L4_Zone1_FWD) ,XIC(LiftZone_FWD) RES(L4_Zone_Timeout[0]) ];
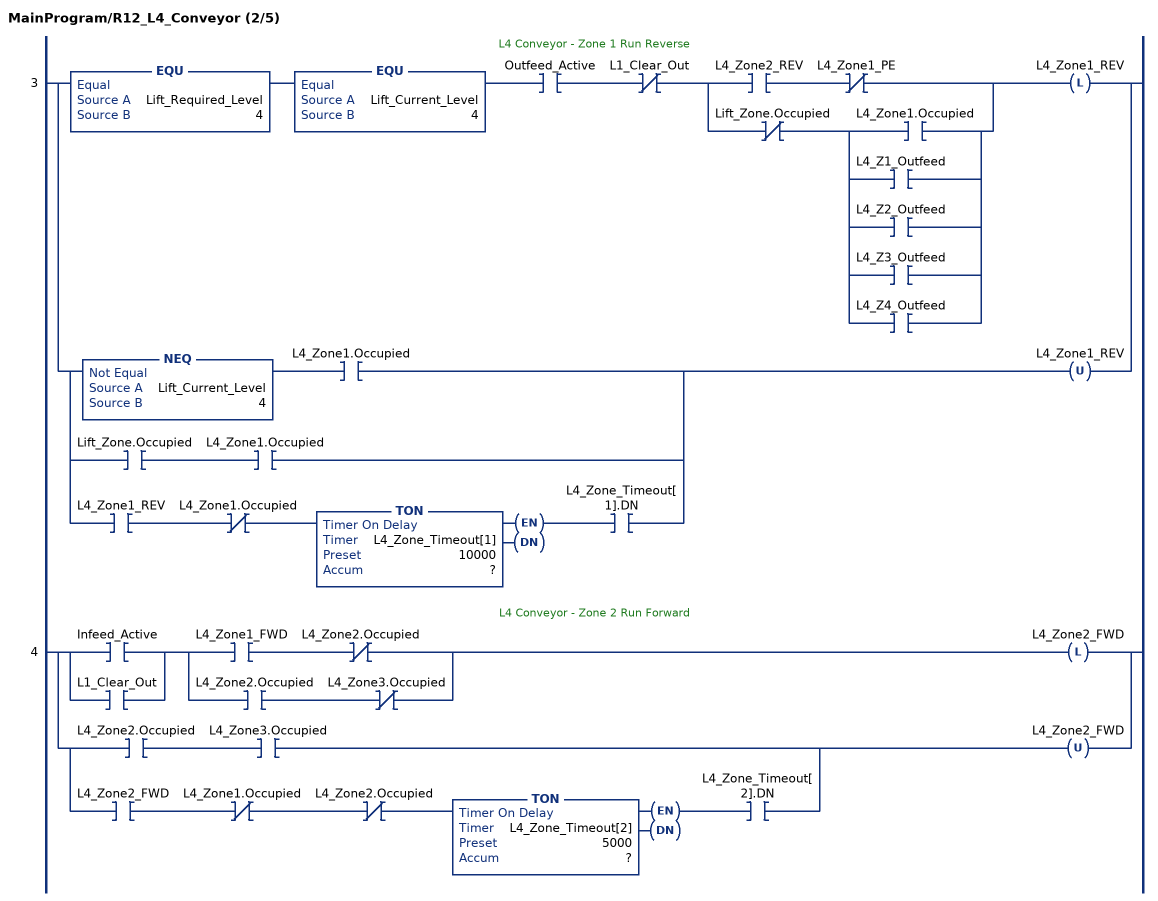
   // L4 Conveyor - Zone 1 Run Reverse
   3: [EQU(Lift_Required_Level,4) EQU(Lift_Current_Level,4) XIC(Outfeed_Active) XIO(L1_Clear_Out) [XIC(L4_Zone2_REV) XIO(L4_Zone1_PE) ,XIO(Lift_Zone.Occupied) [XIC(L4_Zone1.Occupied) ,XIC(L4_Z1_Outfeed) ,XIC(L4_Z2_Outfeed) ,XIC(L4_Z3_Outfeed) ,XIC(L4_Z4_Outfeed) ] ] OTL(L4_Zone1_REV) ,[NEQ(Lift_Current_Level,4) XIC(L4_Zone1.Occupied) ,XIC(Lift_Zone.Occupied) XIC(L4_Zone1.Occupied) ,XIC(L4_Zone1_REV) XIO(L4_Zone1.Occupied) TON(L4_Zone_Timeout[1],?,?) XIC(L4_Zone_Timeout[1].DN) ] OTU(L4_Zone1_REV) ];
   // L4 Conveyor - Zone 2 Run Forward
   4: [[XIC(Infeed_Active) ,XIC(L1_Clear_Out) ] [XIC(L4_Zone1_FWD) XIO(L4_Zone2.Occupied) ,XIC(L4_Zone2.Occupied) XIO(L4_Zone3.Occupied) ] OTL(L4_Zone2_FWD) ,[XIC(L4_Zone2.Occupied) XIC(L4_Zone3.Occupied) ,XIC(L4_Zone2_FWD) XIO(L4_Zone1.Occupied) XIO(L4_Zone2.Occupied) TON(L4_Zone_Timeout[2],?,?) XIC(L4_Zone_Timeout[2].DN) ] OTU(L4_Zone2_FWD) ];
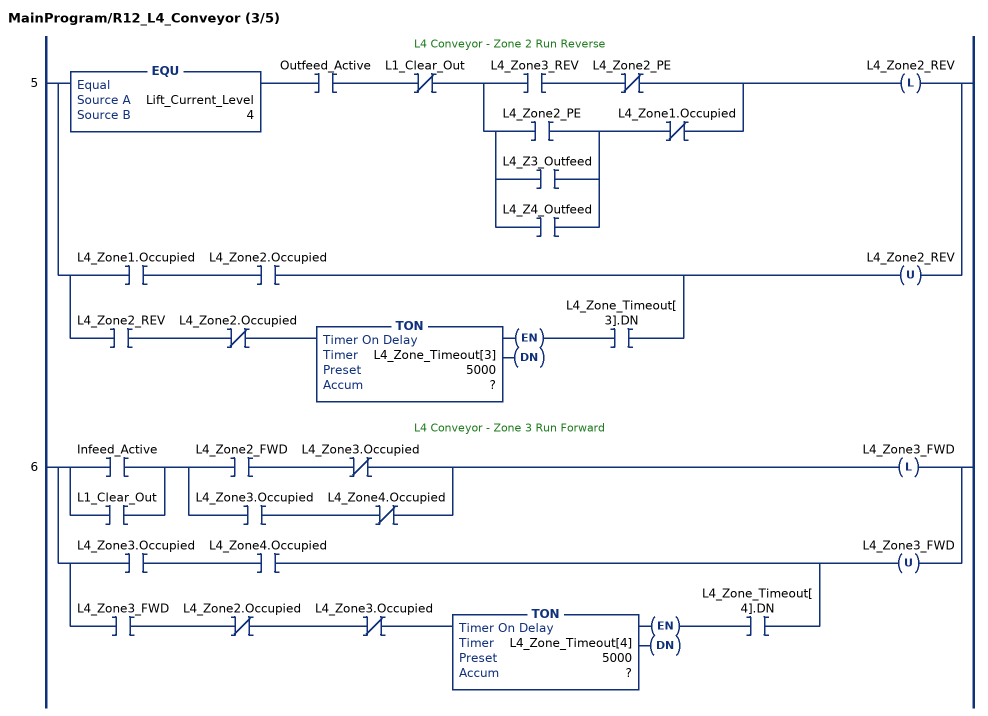
   // L4 Conveyor - Zone 2 Run Reverse
   5: [EQU(Lift_Current_Level,4) XIC(Outfeed_Active) XIO(L1_Clear_Out) [XIC(L4_Zone3_REV) XIO(L4_Zone2_PE) ,[XIC(L4_Zone2_PE) ,XIC(L4_Z3_Outfeed) ,XIC(L4_Z4_Outfeed) ] XIO(L4_Zone1.Occupied) ] OTL(L4_Zone2_REV) ,[XIC(L4_Zone1.Occupied) XIC(L4_Zone2.Occupied) ,XIC(L4_Zone2_REV) XIO(L4_Zone2.Occupied) TON(L4_Zone_Timeout[3],?,?) XIC(L4_Zone_Timeout[3].DN) ] OTU(L4_Zone2_REV) ];
   // L4 Conveyor - Zone 3 Run Forward
   6: [[XIC(Infeed_Active) ,XIC(L1_Clear_Out) ] [XIC(L4_Zone2_FWD) XIO(L4_Zone3.Occupied) ,XIC(L4_Zone3.Occupied) XIO(L4_Zone4.Occupied) ] OTL(L4_Zone3_FWD) ,[XIC(L4_Zone3.Occupied) XIC(L4_Zone4.Occupied) ,XIC(L4_Zone3_FWD) XIO(L4_Zone2.Occupied) XIO(L4_Zone3.Occupied) TON(L4_Zone_Timeout[4],?,?) XIC(L4_Zone_Timeout[4].DN) ] OTU(L4_Zone3_FWD) ];
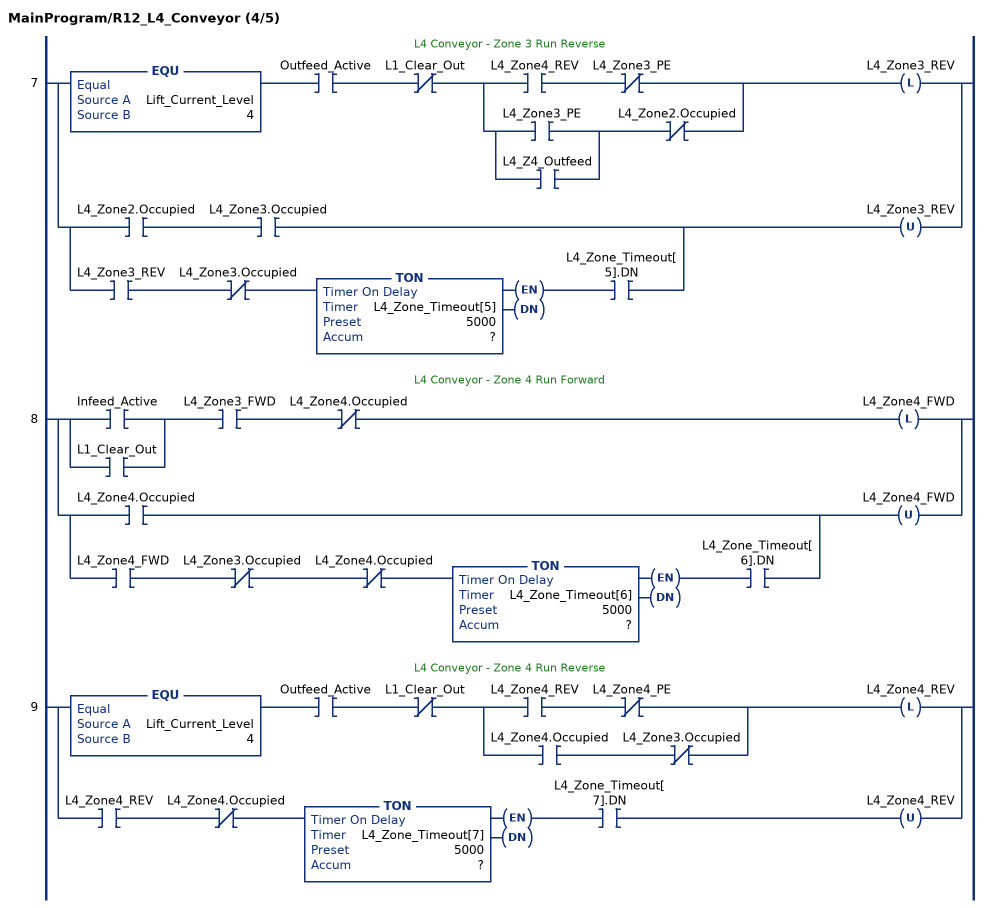
   // L4 Conveyor - Zone 3 Run Reverse
   7: [EQU(Lift_Current_Level,4) XIC(Outfeed_Active) XIO(L1_Clear_Out) [XIC(L4_Zone4_REV) XIO(L4_Zone3_PE) ,[XIC(L4_Zone3_PE) ,XIC(L4_Z4_Outfeed) ] XIO(L4_Zone2.Occupied) ] OTL(L4_Zone3_REV) ,[XIC(L4_Zone2.Occupied) XIC(L4_Zone3.Occupied) ,XIC(L4_Zone3_REV) XIO(L4_Zone3.Occupied) TON(L4_Zone_Timeout[5],?,?) XIC(L4_Zone_Timeout[5].DN) ] OTU(L4_Zone3_REV) ];
   // L4 Conveyor - Zone 4 Run Forward
   8: [[XIC(Infeed_Active) ,XIC(L1_Clear_Out) ] XIC(L4_Zone3_FWD) XIO(L4_Zone4.Occupied) OTL(L4_Zone4_FWD) ,[XIC(L4_Zone4.Occupied) ,XIC(L4_Zone4_FWD) XIO(L4_Zone3.Occupied) XIO(L4_Zone4.Occupied) TON(L4_Zone_Timeout[6],?,?) XIC(L4_Zone_Timeout[6].DN) ] OTU(L4_Zone4_FWD) ];
   // L4 Conveyor - Zone 4 Run Reverse
   9: [EQU(Lift_Current_Level,4) XIC(Outfeed_Active) XIO(L1_Clear_Out) [XIC(L4_Zone4_REV) XIO(L4_Zone4_PE) ,XIC(L4_Zone4.Occupied) XIO(L4_Zone3.Occupied) ] OTL(L4_Zone4_REV) ,XIC(L4_Zone4_REV) XIO(L4_Zone4.Occupied) TON(L4_Zone_Timeout[7],?,?) XIC(L4_Zone_Timeout[7].DN) OTU(L4_Zone4_REV) ];
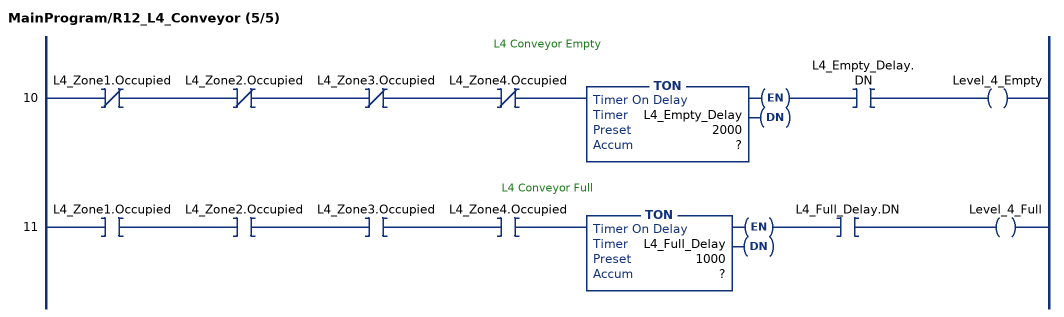
   // L4 Conveyor Empty
   10: XIO(L4_Zone1.Occupied)XIO(L4_Zone2.Occupied)XIO(L4_Zone3.Occupied)XIO(L4_Zone4.Occupied)TON(L4_Empty_Delay,?,?)XIC(L4_Empty_Delay.DN)OTE(Level_4_Empty);
   // L4 Conveyor Full
   11: XIC(L4_Zone1.Occupied)XIC(L4_Zone2.Occupied)XIC(L4_Zone3.Occupied)XIC(L4_Zone4.Occupied)TON(L4_Full_Delay,?,?)XIC(L4_Full_Delay.DN)OTE(Level_4_Full);
END_ROUTINE
